Fanuc KAREL source: KA00223.KL

PROGRAM KA00223
%NOLOCKGROUP
VAR
  SRC: ARRAY[4] OF JOINTPOS
  DST: ARRAY[4] OF VECTOR
BEGIN
  DST = SRC
END KA00223
